// Mitsubishi GX Works2 project: 상승하강펄스   PLC: Q02/Q02H

PROGRAM MAIN
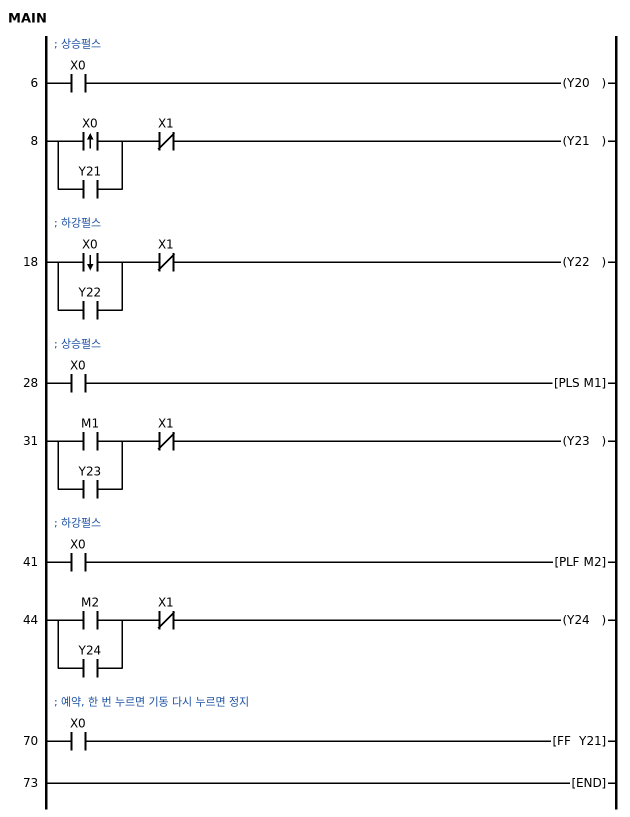
; 상승펄스
6     LD      X0
      OUT     Y20
8     LDP     X0
      OR      Y21
      ANI     X1
      OUT     Y21
; 하강펄스
18    LDF     X0
      OR      Y22
      ANI     X1
      OUT     Y22
; 상승펄스
28    LD      X0
      PLS     M1
31    LD      M1
      OR      Y23
      ANI     X1
      OUT     Y23
; 하강펄스
41    LD      X0
      PLF     M2
44    LD      M2
      OR      Y24
      ANI     X1
      OUT     Y24
; 예약, 한 번 누르면 기동 다시 누르면 정지
70    LD      X0
      FF      Y21
73    END
END_PROGRAM
